Fanuc KAREL source: ko00067.KL

-- PROVISIONAL review KL for V940-1; original PC SHA256 c3b7c00594180eecfa3647c8d8c7325014e23abc4103c079c9117e70b143a20c
-- Incomplete behavior may be omitted. Consult companion uncertainty JSON. Do not deploy.
PROGRAM KO00067
%NOLOCKGROUP
BEGIN
  -- V9_ZERO_TABLE_METADATA_HINT layout=0002_ascii; no indexed target words; source/name/runtime held
  -- UNRESOLVED_PC offsets 5-12; opcodes 9D,23
  -- UNRESOLVED_PC offsets 17-63; opcodes 27,22,1C,22,1C,22,31,7E,4A
  -- UNRESOLVED_PC offsets 68-72; opcodes 7F
END KO00067
